{attribute 'qualified_only'}
{attribute 'strict'}
TYPE E_XYOrientation :
(
	X,
	Y
)USINT;
END_TYPE

(* stored: Version 1.1.0.1, ProductVersion 3.1.4020.12
   DUT E_XYOrientation: Id {87731299-5503-4d18-8225-6c2aff231533} *)
